// TIA Portal V17 export
// export: Created 2025-03-07T09:19:56.2226565Z, ExportSetting WithDefaults, DisplayName Totally Integrated Automation Portal, DisplayVersion V17 Update 8, DisplayName TIA Portal Openness, DisplayVersion V17 Update 8, DisplayName TIA Portal Version Control Interface, DisplayVersion V17, DisplayName SINAMICS Startdrive Advanced, DisplayVersion V17 SP2, DisplayName SINAMICS Startdrive G110M, G120, G120C, G120D, G120P, G115D, DisplayVersion V17 SP2, DisplayName SINAMICS Startdrive G130, G150, S120, S150, SINAMICS MV, S210, DisplayVersion V17 SP2, DisplayName STEP 7 Professional, DisplayVersion V17 Update 8, DisplayName SINUMERIK ONE STEP 7 Toolbox, DisplayVersion V17 Update 12, DisplayName SINUMERIK 840D sl STEP 7 Toolbox, DisplayVersion V17 Update 12, DisplayName STEP 7 Safety, DisplayVersion V17 Update 6, DisplayName WinCC Advanced, DisplayVersion V17 Update 8
TYPE "ROBOT_GRIPPER"
// stored: IsFailsafeCompliant false
   STRUCT
      CLOSED_1_I : Bool;   // CLOSED 1 INPUT
      CLOSED_2_I : Bool;   // CLOSED 2 INPUT
      OPEN_1_I : Bool;   // OPEN 1 INPUT
      OPEN_2_I : Bool;   // OPEN 2 INPUT
      GENERAL_CONDITIONS : Bool;   // GENERAL CONDITIONS
      CLOSE_CONDITIONS : Bool;   // CLOSE CONDITIONS
      OPEN_CONDITIONS : Bool;   // OPEN CONDITIONS
      GENERAL_CONDITIONS_HELP : Bool;   // GENERAL CONDITIONS HELP
      CLOSE_CONDITIONS_HELP : Bool;   // CLOSE CONDITIONS HELP
      OPEN_CONDITIONS_HELP : Bool;   // OPEN CONDITIONS HELP
      HMI_CLOSE_MAN_REQUEST : Bool;   // HMI CLOSE MANUAL REQUEST
      HMI_CLOSE_INDPNDT_MAN_REQUEST : Bool;   // HMI CLOSE INDPNDT MANUAL REQUEST
      CLOSE_MANUAL_REQUEST : Bool;   // CLOSE MANUAL REQUEST
      HMI_OPEN_MAN_REQUEST : Bool;   // HMI OPEN MANUAL REQUEST
      HMI_OPEN_INDPNDT_MAN_REQUEST : Bool;   // HMI OPEN INDPNDT MANUAL REQUEST
      OPEN_MANUAL_REQUEST : Bool;   // OPEN MANUAL REQUEST
      CLOSE_AUTO_REQUEST : Bool;   // CLOSE AUTO REQUEST / CLOSE AUTOMATIC REQUEST
      OPEN_AUTO_REQUEST : Bool;   // OPEN AUTO REQUEST / OPEN AUTOMATIC REQUEST
      CLOSE_GLOBAL_REQUEST : Bool;   // CLOSE GLOBAL REQUEST
      OPEN_GLOBAL_REQUEST : Bool;   // OPEN GLOBAL REQUEST
      CLOSE_COMMAND : Bool;   // CLOSE COMMAND
      OPEN_COMMAND : Bool;   // OPEN COMMAND
      GENERAL_COND_HELP : Bool;   // GENERAL CONDITION HELP
      SIMULTANEITY_FAULT : Bool;   // SIMULTANEITY FAULT
      TIME_EXCEEDED : Bool;   // TIME EXCEEDED
      ALARM : Bool;   // FAULT / ALARM
      PULSE_1 : Bool;   // PULSE 1
      PULSE_2 : Bool;   // PULSE 2
      PULSE_3 : Bool;   // PULSE 3
      AUX_1 : Bool;   // AUXILIARY 1 / AUX 1
      AUX_2 : Bool;   // AUXILIARY 2 / AUX 2
      AUX_3 : Bool;   // AUXILIARY 3 / AUX 3
      AUX_4 : Bool;   // AUXILIARY 4 / AUX 4
   END_STRUCT;
END_TYPE
